PROGRAM PRG_01_Reel
VAR
	TOF_XdriveDelay: TOF;
END_VAR

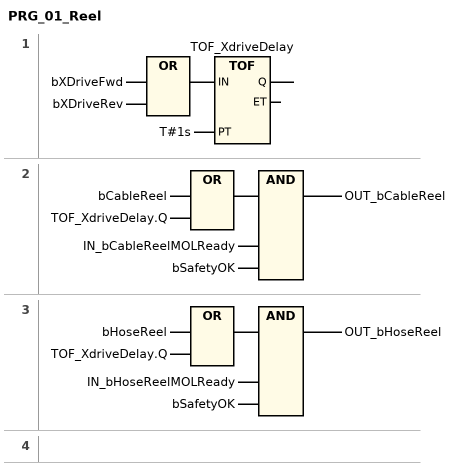
// NETWORK 1
TOF_XdriveDelay(IN := bXDriveFwd OR bXDriveRev, PT := T#1s); // TOF

// NETWORK 2
OUT_bCableReel := (bCableReel OR TOF_XdriveDelay.Q) AND IN_bCableReelMOLReady AND bSafetyOK;

// NETWORK 3
OUT_bHoseReel := (bHoseReel OR TOF_XdriveDelay.Q) AND IN_bHoseReelMOLReady AND bSafetyOK;

// NETWORK 4

END_PROGRAM

(* stored: Version 1.1.0.1, ProductVersion 3.1.4024.15
   POU PRG_01_Reel: Id {5e03e5ee-3757-4033-b590-e328a09ccb5c}, SpecialFunc None *)
